// Mitsubishi GX Works2 project: 26 unfinish   PLC: FX3G

// task Task_01 (event TRUE, interval 0, priority 31): POU_01

PROGRAM POU_01
VAR
  gas : INT;
  gas2 : INT;
  ii : INT;
  ton1 : TON;
  ton2 : TON;
  ton3 : TON;
  ton4 : TON;
  ton5 : TON;
  ton6 : TON;
  ton7 : TON;
  ton8 : TON;
  rf1 : R_TRIG;
END_VAR
IF M8002 THEN
	gas := 0;
END_IF;

IF M4 THEN
	
	gas:=99;
END_IF;


CASE gas OF
	0:
	IF M5 THEN
		gas:=1;
	END_IF;
	
	1:
	Y3:=TRUE;
	Y5:=TRUE;
	Y2:=FALSE;
	ton1(IN := NOT ton1.Q, PT := T#8s);
	IF ton1.Q THEN
		gas:=2;
	END_IF;
	
	2:
	Y3:=M8013;
	ton2(IN := NOT ton2.Q, PT := T#3s);
	IF ton2.Q THEN
		gas:=3;
	END_IF;
	
	3:
	Y3:=FALSE;
	Y4:=TRUE;
	ton3(IN := NOT ton3.Q, PT := T#3s);
	IF ton3.Q THEN
		gas:=4;
	END_IF;

 	4:
 	Y4:=FALSE;
 	Y5:=FALSE;
 		ton4(IN := NOT ton4.Q, PT := T#0.5s);
	IF ton4.Q THEN
		gas:=5;
	END_IF;
	
	5:
 Y2:=TRUE;
 Y0:=TRUE;
 ton5(IN := NOT ton5.Q, PT := T#8s);
	IF ton5.Q THEN
		gas:=6;
	END_IF;
	
	6:
	Y0:=M8013;
	ton6(IN := NOT ton6.Q, PT := T#3s);
	IF ton6.Q THEN
		gas:=7;
	END_IF;
	
	7:
	Y0:=FALSE;
	Y1:=TRUE;
	ton7(IN := NOT ton7.Q, PT := T#3s);
	IF ton7.Q THEN
		gas:=8;
	END_IF;

	8:
	Y1:=FALSE;
	Y2:=TRUE;
	ton8(IN := NOT ton8.Q, PT := T#0.5s);
	IF ton8.Q THEN
		gas:=1;
	END_IF;

	99:
	Y4:=M8013;
	Y1:=M8013;
	Y2:=FALSE;
	Y3:=FALSE;
	Y5:=FALSE;
	
		IF NOT M4 THEN
			gas:=1;
		END_IF;
		

END_CASE;
END_PROGRAM
